Universal Robots PolyScope program: Socket_test4.urp

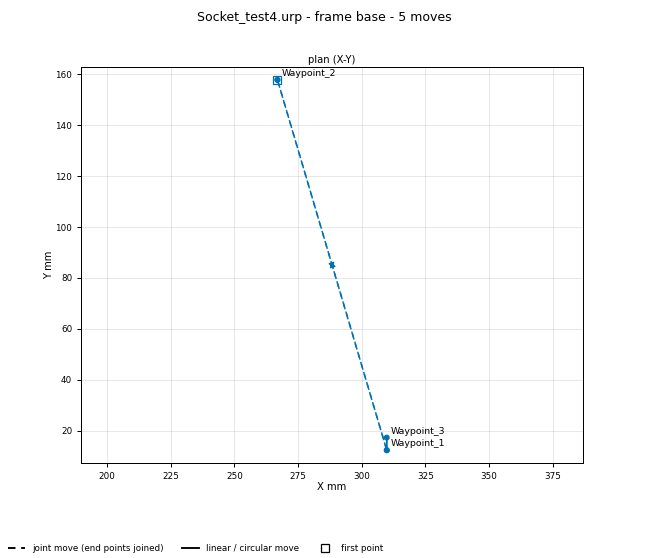
[picture p0: tool path of Socket_test4.urp in frame base, 5 of 5 moves have a stored position in this frame; points joined in program order, loops and branches not executed]
ProgramRoot directory=/programs/KSJ; kinematics=(a=[0.00002, -0.60789, -0.56786, -0.00004, 0.00004, 0], d=[0.12818, 49.57086, -69.93345, 20.52608, 0.11576, 0.09196], alpha=[1.57118, -0.00157, -0.00317, 1.57037, -1.57091, 0], deltaTheta=[-0.00001, -0.12723, 0.24046, -0.11324, -0.00006, 0.00005], status=notLinearised); lastSavedInVersion=(project__name=Polyscope, major__version=3, minor__version=1, svn__revision=16916, build__date=Feb 06 2015, 15:15:00); name=Socket_test4; programVersion=(project__name=Polyscope, major__version=3, minor__version=0, svn__revision=16471, build__date=Dec 02 2014, 09:52:01); robotEnvironmentFileName=Fomeco_1; serialNumberRobot=2014300380
  BeforeStart description=COMMAND_SEQUENCE_BEFORE_PROGRAM_START; name=BeforeStart
    Script type=1; cachedFileContents=#Activation if not activated
      | if ((modbus_get_signal_status("Gripper_Status1", False) == False)  and (modbus_get_signal_status("Gripper_Status2", False) == False)):
      |     modbus_set_output_signal("Activate", True, False)
      | end
      | 
      | #Prohibit the movement
      | modbus_set_output_signal("Go_to_Requested", False, False)
      | while (modbus_get_signal_status("Action_Status", False) == True):
      |     sync()
      | end
      | 
      | #Awaiting the activation of the gripper
      | while (not(modbus_get_signal_status("Gripper_Status1", False) ==  True )):
      |     sync()
      | end
      | while (not(modbus_get_signal_status("Gripper_Status2", False) ==  True )):
      |     sync()
      | end; scriptFile=/programs/RQ_2FG_Activate_script.script
    Assignment expr="192.168.2.14"; operatorValueType=INTEGER; valueSource=EXPRESSION
    Assignment expr=30000; operatorValueType=INTEGER; valueSource=EXPRESSION
    Assignment expr="test"; operatorValueType=INTEGER; valueSource=EXPRESSION
    Assignment expr=1; operatorValueType=INTEGER; valueSource=EXPRESSION
    Assignment expr=socket_open(socket_ip,socket_port, socket_name); operatorValueType=INTEGER; valueSource=EXPRESSION
    Move cartesianAcceleration=1.2; cartesianSpeed=0.25; jointAcceleration=1.3962634015954636; jointSpeed=1.0471975511965976; sharedProcessMoveBlendRadius=0.025; motionType=JOINT_SPACE
      Waypoint blendRadius=0.05; cartesianAcceleration=1.2; cartesianSpeed=0.25; jointAcceleration=1.3962634015954636; jointSpeed=1.0471975511965976; nextMotionTime=2.0; stoppoint=true; useSharedBlendParameter=true; useSharedParameters=true; position=TCP in base x=266.893 y=157.817 z=473.548 mm, rx=2.7028 ry=-1.5985 rz=0.0143 rad; joints [57.388, -57.249, -103.899, -108.909, 89.333, 28.719] deg; positionType=FIXED_POSITION; waypointPoseInFeatureCoordinates=(pos=(x=0.26689302408305, y=0.15781699190306892, z=0.47354802210578134), rot=(x=2.7028242999956396, y=-1.5985155770946289, z=0.014274333770486309)); name=Waypoint_2
    While count=0; expr=ExpressionVariableNode≟ False; type=LOOP_EXPR
      Assignment expr=socket_open(socket_ip, socket_port, socket_name); operatorValueType=INTEGER; valueSource=EXPRESSION
      Wait 
    Move cartesianAcceleration=1.2; cartesianSpeed=0.25; jointAcceleration=1.3962634015954636; jointSpeed=1.0471975511965976; sharedProcessMoveBlendRadius=0.025; motionType=JOINT_SPACE
      Waypoint blendRadius=0.05; cartesianAcceleration=1.2; cartesianSpeed=0.25; jointAcceleration=1.3962634015954636; jointSpeed=1.0471975511965976; nextMotionTime=2.0; stoppoint=true; useSharedBlendParameter=true; useSharedParameters=true; position=TCP in base x=309.828 y=12.339 z=473.571 mm, rx=2.2301 ry=-2.207 rz=0.0102 rad; joints [28.975, -57.309, -103.868, -108.929, 89.438, 28.51] deg; positionType=FIXED_POSITION; waypointPoseInFeatureCoordinates=(pos=(x=0.3098282101263387, y=0.012339393940506063, z=0.47357122952219893), rot=(x=2.2301324054852167, y=-2.2069823580211625, z=0.010169530319051826)); name=Waypoint_1
    Assignment expr=get_actual_tcp_pose(); operatorValueType=INTEGER; valueSource=EXPRESSION
  SubProgram [hidden by the author, left out]
  SubProgram [hidden by the author, left out]
  MainProgram cartesianAcceleration=1.2; cartesianSpeed=0.25; jointAcceleration=1.3962634015954636; jointSpeed=1.0471975511965976; sharedProcessMoveBlendRadius=0.025; motionType=JOINT_SPACE; runOnlyOneCycle=true
    Script type=0; expressionBranchNode=socket_send_string(ExpressionVariableNode, socket_name)
    Suppressed suppressedNode=(waitTime=1.0)
    Assignment expr=socket_read_ascii_float(5, socket_name); operatorValueType=INTEGER; valueSource=EXPRESSION
    Suppressed suppressedNode=ExpressionVariableNode[0]≟0
    If expr=ExpressionVariableNode[0]≠0; type=IF_NODE
      Assignment expr=-var_2[1]; operatorValueType=INTEGER; valueSource=EXPRESSION
      Assignment expr=-ExpressionVariableNode[2]; operatorValueType=INTEGER; valueSource=EXPRESSION
      Assignment expr=-ExpressionVariableNode[3]; operatorValueType=INTEGER; valueSource=EXPRESSION
      Assignment expr=ExpressionVariableNode[4]; operatorValueType=INTEGER; valueSource=EXPRESSION
      Assignment expr=var_2[5]; operatorValueType=INTEGER; valueSource=EXPRESSION
      Assignment expr=0; operatorValueType=INTEGER; valueSource=EXPRESSION
      Assignment expr=p[ExpressionVariableNode, 0, ExpressionVariableNode, 0, 0, 0]; operatorValueType=INTEGER; valueSource=EXPRESSION
      Assignment expr=p[naaldafstand,0 ,0 ,0 ,0 ,0]; operatorValueType=INTEGER; valueSource=EXPRESSION
      Assignment expr=pose_trans(ExpressionVariableNode, ExpressionVariableNode); operatorValueType=INTEGER; valueSource=EXPRESSION
      Assignment expr=ExpressionVariableNode; operatorValueType=INTEGER; valueSource=EXPRESSION
      Move cartesianAcceleration=1.2; cartesianSpeed=0.25; jointAcceleration=1.3962634015954636; jointSpeed=1.0471975511965976; sharedProcessMoveBlendRadius=0.025; motionType=CARTESIAN_SPACE
        Waypoint blendRadius=0.05; cartesianAcceleration=1.2; cartesianSpeed=0.25; jointAcceleration=1.3962634015954636; jointSpeed=1.0471975511965976; nextMotionTime=2.0; stoppoint=true; useSharedBlendParameter=true; useSharedParameters=true; positionType=VARIABLE_POSITION; name=Waypoint
      While count=0; expr=ctr1<ExpressionVariableNode; type=LOOP_EXPR
        Move cartesianAcceleration=1.2; cartesianSpeed=0.25; jointAcceleration=1.3962634015954636; jointSpeed=1.0471975511965976; sharedProcessMoveBlendRadius=0.025; motionType=CARTESIAN_SPACE
          Waypoint blendRadius=0.05; cartesianAcceleration=1.2; cartesianSpeed=0.25; jointAcceleration=1.3962634015954636; jointSpeed=1.0471975511965976; nextMotionTime=2.0; stoppoint=true; useSharedBlendParameter=true; useSharedParameters=true; position=TCP in base x=309.811 y=17.315 z=473.615 mm, rx=2.2301 ry=-2.2072 rz=0.0102 rad; joints [29.74, -57.335, -103.859, -108.919, 89.438, 29.276] deg; positionType=VARIABLE_POSITION; waypointPoseInFeatureCoordinates=(pos=(x=0.3098112575352612, y=0.01731501006793316, z=0.4736149848983391), rot=(x=2.230071758870465, y=-2.2071749142722723, z=0.01021593393263643)); name=Waypoint_3
        Assignment expr=get_actual_tcp_pose(); operatorValueType=INTEGER; valueSource=EXPRESSION
        Assignment expr=pose_trans(ExpressionVariableNode,p_nextx); operatorValueType=INTEGER; valueSource=EXPRESSION
        Wait 
        Assignment expr=ExpressionVariableNode+1; operatorValueType=INTEGER; valueSource=EXPRESSION
      Move cartesianAcceleration=1.2; cartesianSpeed=0.25; jointAcceleration=1.3962634015954636; jointSpeed=1.0471975511965976; sharedProcessMoveBlendRadius=0.025; motionType=CARTESIAN_SPACE
        Waypoint blendRadius=0.05; cartesianAcceleration=1.2; cartesianSpeed=0.25; jointAcceleration=1.3962634015954636; jointSpeed=1.0471975511965976; nextMotionTime=2.0; stoppoint=true; useSharedBlendParameter=true; useSharedParameters=true; outputFlangePose=(pos=(x=0.36432781318860386, y=0.015104207999906234, z=0.7357060438895484), rot=(x=2.230185760310772, y=-2.2070852141972783, z=0.010116155461847413)); position=TCP in base x=309.828 y=12.339 z=473.571 mm, rx=2.2301 ry=-2.207 rz=0.0102 rad; joints [28.975, -57.309, -103.868, -108.929, 89.438, 28.51] deg; positionType=FIXED_POSITION; waypointPoseInFeatureCoordinates=(pos=(x=0.3098282101263387, y=0.012339393940506063, z=0.47357122952219893), rot=(x=2.2301324054852167, y=-2.2069823580211625, z=0.010169530319051826)); name=Waypoint_1
      Move cartesianAcceleration=1.2; cartesianSpeed=0.25; jointAcceleration=1.3962634015954636; jointSpeed=1.0471975511965976; sharedProcessMoveBlendRadius=0.025; motionType=JOINT_SPACE
        Waypoint blendRadius=0.05; cartesianAcceleration=1.2; cartesianSpeed=0.25; jointAcceleration=1.3962634015954636; jointSpeed=1.0471975511965976; nextMotionTime=2.0; stoppoint=true; useSharedBlendParameter=true; useSharedParameters=true; position=TCP in base x=266.893 y=157.817 z=473.548 mm, rx=2.7028 ry=-1.5985 rz=0.0143 rad; joints [57.388, -57.249, -103.899, -108.909, 89.333, 28.719] deg; positionType=FIXED_POSITION; waypointPoseInFeatureCoordinates=(pos=(x=0.26689302408305, y=0.15781699190306892, z=0.47354802210578134), rot=(x=2.7028242999956396, y=-1.5985155770946289, z=0.014274333770486309)); name=Waypoint_2
      Suppressed suppressedNode=(CallSubProgramNode=(default=(subProgramNodeToCall=0)))
      Suppressed suppressedNode=(CallSubProgramNode=(default=(subProgramNodeToCall=255)))
